// TIA Portal V20 export
TYPE "UDT_Interlock_manual_AMR"
   STRUCT
      "byte0.bit0" : Bool;
      "byte0.bit1" : Bool;
      "byte0.bit2" : Bool;
      "byte0.bit3" : Bool;
      "byte0.bit4" : Bool;
      "Byte0.bit5" : Bool;
      "Byte0.bit6" : Bool;
      Drop_Enable : Bool;
      Byte1_bit0 : Bool;
      Byte1_bit1 : Bool;
      Byte1_bit2 : Bool;
      Byte1_bit3 : Bool;
      Byte1_bit4 : Bool;
      Byte1_bit5 : Bool;
      Byte1_bit6 : Bool;
      Pick_Enable : Bool;
   END_STRUCT;
END_TYPE
